FUNCTION_BLOCK FB_DeviceByte EXTENDS FB_LinkDataByte
VAR_INPUT		
	nControl  			: BYTE;
	nControlData  		: BYTE;
END_VAR

VAR_OUTPUT
	nStatus  			: BYTE;
	nStatusData  		: BYTE;
END_VAR

SUPER^();
Control := nControl;
ControlData := nControlData;
nStatus := Status;
nStatusData := StatusData;

END_FUNCTION_BLOCK

(* stored: Version 1.1.0.1, ProductVersion 3.1.4024.12
   POU FB_DeviceByte: Id {1ebe7cac-dcf7-002d-235a-1745320b2e41}, SpecialFunc None *)
